{attribute 'GeneratedUsingTerminal: EK1122-0000-0018'}
{attribute addProperty BoxType "EK1122-0000-0018"}
{attribute addProperty Id "A_0060_AT2020_0250_0019_AT2020_0250A_0060_AT2020_0250_0019_AT2020_0250_29EE827680Beckhoff_AT2xxxsub_EK1100EK1100_1FC0878B2A_0001_AT2000_0233_0022AT2000_1809CD2F80A_0002_AT2000_0233_0023AT2000_1809CD2F80A_0003_AT2000_0233_0024AT2000_1809CD2F80A_0004_AT2000_0250_0016AT2000_2EA6C9BF84A_0005_AT2000_0250_0017AT2000_2EA6C9BF84A_0006_AT2000_0250_0018AT2000_2EA6C9BF84A_0007_AT2000_0250_0019AT2000_2EA6C9BF84A_0008_AT2000_0250_0020AT2000_2EA6C9BF84A_0009_AT2000_0250_0021AT2000_2EA6C9BF84A_0010_AT2000_0250_0022AT2000_2EA6C9BF84A_0011_AT2000_0250_0023AT2000_2EA6C9BF84A_0012_AT2001_0250_0016AT2001_2EA6C9BF84A_0013_AT2001_0250_0017AT2001_2EA6C9BF84A_0014_AT2001_0250_0018AT2001_2EA6C9BF84A_0015_AT2001_0250_0019AT2001_2EA6C9BF84A_0016_AT2001_0250_0020AT2001_2EA6C9BF84A_0017_AT2001_0250_0022AT2001_2EA6C9BF84A_0018_AT2001_0250_0023AT2001_2EA6C9BF84A_0019_AT2001_0250_0024AT2001_2EA6C9BF84A_0020_AT2002_0249_0021AT2002_2EA6C9BF84A_0021_AT2002_0249_0022AT2002_2EA6C9BF84A_0022_AT2002_0249_0023AT2002_2EA6C9BF84A_0023_AT2002_0250_0022AT2002_2EA6C9BF84A_0024_AT2002_0250_0023AT2002_2EA6C9BF84A_0025_AT2002_0250_0024AT2002_2EA6C9BF84A_0026_AT2020_0250_0018AT2020_2EA6C9BF84A_0027_AT2020_0250_0021AT2020_2EA6C9BF84A_0028_AT2021_0250_0018AT2021_2EA6C9BF84A_0029_AT2021_0250_0020AT2021_2EA6C9BF84A_0030_AT2025_0250_0018AT2025_2EA6C9BF84A_0031_AT2026_0250_0021AT2026_2EA6C9BF84A_0032_AT2026_0250_0023AT2026_2EA6C9BF84A_0033_AT2040_0250_0018AT2040_2EA6C9BF84A_0034_AT2040_0250_0019AT2040_2EA6C9BF84A_0035_AT2040_0250_0020AT2040_2EA6C9BF84A_0036_AT2040_0250_0021A_0036_AT2040_0250_0021_0B822AE480A_0037_AT2040_0250_0022A_0037_AT2040_0250_0022_033DCEC480A_0038_AT2040_0250_0023A_0038_AT2040_0250_0023_C339CA0C80A_0039_AT2040_0250_0024A_0039_AT2040_0250_0024_375958EA80A_0040_AT2041_0250_0018A_0040_AT2041_0250_0018_536500F280A_0041_AT2041_0250_0019A_0041_AT2041_0250_0019_F34F405680A_0042_AT2041_0250_0020A_0042_AT2041_0250_0020_5E65A51E80A_0043_AT2041_0250_0021A_0043_AT2041_0250_0021_AA0537F880A_0044_AT2041_0250_0022A_0044_AT2041_0250_0022_5A9A39BA80A_0045_AT2041_0250_0023A_0045_AT2041_0250_0023_51C662AC80A_0046_AT2042_0250_0024A_0046_AT2042_0250_0024_1B20CF3180A_0047_AT2050_0500_0016A_0047_AT2050_0500_0016_139F2B1180A_0048_AT2050_0500_0017A_0048_AT2050_0500_0017_3F977F4780A_0049_AT2050_0500_0018A_0049_AT2050_0500_0018_CBE655A880A_0050_AT2050_0500_0019A_0050_AT2050_0500_0019_15A3AE6F80A_0051_AT2050_0500_0020A_0051_AT2050_0500_0020_9B531B4E80A_0052_AT2050_0500_0021A_0052_AT2050_0500_0021_4516E08980A_0053_AT2050_0500_0022A_0053_AT2050_0500_0022_433BDDFE80A_0054_AT2050_0500_0023A_0054_AT2050_0500_0023_B2F2DF5580A_0055_AT2050_0500_0024A_0055_AT2050_0500_0024_8D42A08D80A_0056_AT2050_0501_0017A_0056_AT2050_0501_0017_A14AF4DB80A_0057_AT2050_0501_0020A_0057_AT2050_0501_0020_A9F510FB80A_0058_AT2050_0501_0021A_0058_AT2050_0501_0021_DD8E109080A_0061_AT2020_0250_0023_AT2020_0250A_0061_AT2020_0250_0023_AT2020_0250_2D9AB3DC80A_0062_AT2025_0250_0020_AT2025_0250A_0062_AT2025_0250_0020_AT2025_0250_8DB0F37880A_0063_AT2025_0250_0022_AT2025_0250A_0063_AT2025_0250_0022_AT2025_0250_E88F66A280A_0064_AT2025_0250_0023_AT2025_0250A_0064_AT2025_0250_0023_AT2025_0250_894F6FDC80A_0065_AT2026_0250_0019_AT2026_0250A_0065_AT2026_0250_0019_AT2026_0250_A5473B8A80A_0066_AT2026_0250_0020_AT2026_0250A_0066_AT2026_0250_0020_AT2026_0250_ADF8DFAA80A_0067_AT2026_0250_0022_AT2026_0250A_0067_AT2026_0250_0022_AT2026_0250_BF728FE680A_0068_AT2026_0250_0024_AT2026_0250A_0068_AT2026_0250_0024_AT2026_0250_71C0116580A_0069_AT2050_0501_0019_AT2050_0501A_0069_AT2050_0501_0019_AT2050_0501_10255FA680A_0070_AT2050_0501_0022_AT2050_0501A_0070_AT2050_0501_0022_AT2050_0501_E445CD4080A_0071_AT2050_0501_0023_AT2050_0501A_0071_AT2050_0501_0023_AT2050_0501_A5CC968480A_0072_AT2050_0501_0024_AT2050_0501A_0072_AT2050_0501_0024_AT2050_0501_05E6D62080"}
{attribute addProperty CRC "1138582487"}
{attribute addProperty Size "5810"}
TYPE Beckhoff_AT2xxxEK1122_43DD63D7 EXTENDS EK1122_1FC0878B :
STRUCT
	{attribute addProperty Name "A_0060_AT2020_0250_0019_AT2020_0250"}
	{attribute addProperty PreviousPort "Beckhoff AT2xxxEK1122 : D"}
	A_0060_AT2020_0250_0019_AT2020_0250 : A_0060_AT2020_0250_0019_AT2020_0250_29EE8276;
	{attribute addProperty Name "Beckhoff_AT2xxxsub_EK1100"}
	{attribute addProperty PreviousPort "A_0060(AT2020-0250-0019) (AT2020-0250) : C"}
	Beckhoff_AT2xxxsub_EK1100 : EK1100_1FC0878B;
	{attribute addProperty Name "A_0001_AT2000_0233_0022"}
	{attribute addProperty PreviousPort "Beckhoff AT2xxxsub EK1100 : C"}
	A_0001_AT2000_0233_0022 : AT2000_1809CD2F;
	{attribute addProperty Name "A_0002_AT2000_0233_0023"}
	{attribute addProperty PreviousPort "A_0001(AT2000-0233-0022) : C"}
	A_0002_AT2000_0233_0023 : AT2000_1809CD2F;
	{attribute addProperty Name "A_0003_AT2000_0233_0024"}
	{attribute addProperty PreviousPort "A_0002(AT2000-0233-0023) : C"}
	A_0003_AT2000_0233_0024 : AT2000_1809CD2F;
	{attribute addProperty Name "A_0004_AT2000_0250_0016"}
	{attribute addProperty PreviousPort "A_0003(AT2000-0233-0024) : C"}
	A_0004_AT2000_0250_0016 : AT2000_2EA6C9BF;
	{attribute addProperty Name "A_0005_AT2000_0250_0017"}
	{attribute addProperty PreviousPort "A_0004(AT2000-0250-0016) : C"}
	A_0005_AT2000_0250_0017 : AT2000_2EA6C9BF;
	{attribute addProperty Name "A_0006_AT2000_0250_0018"}
	{attribute addProperty PreviousPort "A_0005(AT2000-0250-0017) : C"}
	A_0006_AT2000_0250_0018 : AT2000_2EA6C9BF;
	{attribute addProperty Name "A_0007_AT2000_0250_0019"}
	{attribute addProperty PreviousPort "A_0006(AT2000-0250-0018) : C"}
	A_0007_AT2000_0250_0019 : AT2000_2EA6C9BF;
	{attribute addProperty Name "A_0008_AT2000_0250_0020"}
	{attribute addProperty PreviousPort "A_0007(AT2000-0250-0019) : C"}
	A_0008_AT2000_0250_0020 : AT2000_2EA6C9BF;
	{attribute addProperty Name "A_0009_AT2000_0250_0021"}
	{attribute addProperty PreviousPort "A_0008(AT2000-0250-0020) : C"}
	A_0009_AT2000_0250_0021 : AT2000_2EA6C9BF;
	{attribute addProperty Name "A_0010_AT2000_0250_0022"}
	{attribute addProperty PreviousPort "A_0009(AT2000-0250-0021) : C"}
	A_0010_AT2000_0250_0022 : AT2000_2EA6C9BF;
	{attribute addProperty Name "A_0011_AT2000_0250_0023"}
	{attribute addProperty PreviousPort "A_0010(AT2000-0250-0022) : C"}
	A_0011_AT2000_0250_0023 : AT2000_2EA6C9BF;
	{attribute addProperty Name "A_0012_AT2001_0250_0016"}
	{attribute addProperty PreviousPort "A_0011(AT2000-0250-0023) : C"}
	A_0012_AT2001_0250_0016 : AT2001_2EA6C9BF;
	{attribute addProperty Name "A_0013_AT2001_0250_0017"}
	{attribute addProperty PreviousPort "A_0012(AT2001-0250-0016) : C"}
	A_0013_AT2001_0250_0017 : AT2001_2EA6C9BF;
	{attribute addProperty Name "A_0014_AT2001_0250_0018"}
	{attribute addProperty PreviousPort "A_0013(AT2001-0250-0017) : C"}
	A_0014_AT2001_0250_0018 : AT2001_2EA6C9BF;
	{attribute addProperty Name "A_0015_AT2001_0250_0019"}
	{attribute addProperty PreviousPort "A_0014(AT2001-0250-0018) : C"}
	A_0015_AT2001_0250_0019 : AT2001_2EA6C9BF;
	{attribute addProperty Name "A_0016_AT2001_0250_0020"}
	{attribute addProperty PreviousPort "A_0015(AT2001-0250-0019) : C"}
	A_0016_AT2001_0250_0020 : AT2001_2EA6C9BF;
	{attribute addProperty Name "A_0017_AT2001_0250_0022"}
	{attribute addProperty PreviousPort "A_0016(AT2001-0250-0020) : C"}
	A_0017_AT2001_0250_0022 : AT2001_2EA6C9BF;
	{attribute addProperty Name "A_0018_AT2001_0250_0023"}
	{attribute addProperty PreviousPort "A_0017(AT2001-0250-0022) : C"}
	A_0018_AT2001_0250_0023 : AT2001_2EA6C9BF;
	{attribute addProperty Name "A_0019_AT2001_0250_0024"}
	{attribute addProperty PreviousPort "A_0018(AT2001-0250-0023) : C"}
	A_0019_AT2001_0250_0024 : AT2001_2EA6C9BF;
	{attribute addProperty Name "A_0020_AT2002_0249_0021"}
	{attribute addProperty PreviousPort "A_0019(AT2001-0250-0024) : C"}
	A_0020_AT2002_0249_0021 : AT2002_2EA6C9BF;
	{attribute addProperty Name "A_0021_AT2002_0249_0022"}
	{attribute addProperty PreviousPort "A_0020(AT2002-0249-0021) : C"}
	A_0021_AT2002_0249_0022 : AT2002_2EA6C9BF;
	{attribute addProperty Name "A_0022_AT2002_0249_0023"}
	{attribute addProperty PreviousPort "A_0021(AT2002-0249-0022) : C"}
	A_0022_AT2002_0249_0023 : AT2002_2EA6C9BF;
	{attribute addProperty Name "A_0023_AT2002_0250_0022"}
	{attribute addProperty PreviousPort "A_0022(AT2002-0249-0023) : C"}
	A_0023_AT2002_0250_0022 : AT2002_2EA6C9BF;
	{attribute addProperty Name "A_0024_AT2002_0250_0023"}
	{attribute addProperty PreviousPort "A_0023(AT2002-0250-0022) : C"}
	A_0024_AT2002_0250_0023 : AT2002_2EA6C9BF;
	{attribute addProperty Name "A_0025_AT2002_0250_0024"}
	{attribute addProperty PreviousPort "A_0024(AT2002-0250-0023) : C"}
	A_0025_AT2002_0250_0024 : AT2002_2EA6C9BF;
	{attribute addProperty Name "A_0026_AT2020_0250_0018"}
	{attribute addProperty PreviousPort "A_0025(AT2002-0250-0024) : C"}
	A_0026_AT2020_0250_0018 : AT2020_2EA6C9BF;
	{attribute addProperty Name "A_0027_AT2020_0250_0021"}
	{attribute addProperty PreviousPort "A_0026(AT2020-0250-0018) : C"}
	A_0027_AT2020_0250_0021 : AT2020_2EA6C9BF;
	{attribute addProperty Name "A_0028_AT2021_0250_0018"}
	{attribute addProperty PreviousPort "A_0027(AT2020-0250-0021) : C"}
	A_0028_AT2021_0250_0018 : AT2021_2EA6C9BF;
	{attribute addProperty Name "A_0029_AT2021_0250_0020"}
	{attribute addProperty PreviousPort "A_0028(AT2021-0250-0018) : C"}
	A_0029_AT2021_0250_0020 : AT2021_2EA6C9BF;
	{attribute addProperty Name "A_0030_AT2025_0250_0018"}
	{attribute addProperty PreviousPort "A_0029(AT2021-0250-0020) : C"}
	A_0030_AT2025_0250_0018 : AT2025_2EA6C9BF;
	{attribute addProperty Name "A_0031_AT2026_0250_0021"}
	{attribute addProperty PreviousPort "A_0030(AT2025-0250-0018) : C"}
	A_0031_AT2026_0250_0021 : AT2026_2EA6C9BF;
	{attribute addProperty Name "A_0032_AT2026_0250_0023"}
	{attribute addProperty PreviousPort "A_0031(AT2026-0250-0021) : C"}
	A_0032_AT2026_0250_0023 : AT2026_2EA6C9BF;
	{attribute addProperty Name "A_0033_AT2040_0250_0018"}
	{attribute addProperty PreviousPort "A_0032(AT2026-0250-0023) : C"}
	A_0033_AT2040_0250_0018 : AT2040_2EA6C9BF;
	{attribute addProperty Name "A_0034_AT2040_0250_0019"}
	{attribute addProperty PreviousPort "A_0033(AT2040-0250-0018) : C"}
	A_0034_AT2040_0250_0019 : AT2040_2EA6C9BF;
	{attribute addProperty Name "A_0035_AT2040_0250_0020"}
	{attribute addProperty PreviousPort "A_0034(AT2040-0250-0019) : C"}
	A_0035_AT2040_0250_0020 : AT2040_2EA6C9BF;
	{attribute addProperty Name "A_0036_AT2040_0250_0021"}
	{attribute addProperty PreviousPort "A_0035(AT2040-0250-0020) : C"}
	A_0036_AT2040_0250_0021 : A_0036_AT2040_0250_0021_0B822AE4;
	{attribute addProperty Name "A_0037_AT2040_0250_0022"}
	{attribute addProperty PreviousPort "A_0036(AT2040-0250-0021) : C"}
	A_0037_AT2040_0250_0022 : A_0037_AT2040_0250_0022_033DCEC4;
	{attribute addProperty Name "A_0038_AT2040_0250_0023"}
	{attribute addProperty PreviousPort "A_0037(AT2040-0250-0022) : C"}
	A_0038_AT2040_0250_0023 : A_0038_AT2040_0250_0023_C339CA0C;
	{attribute addProperty Name "A_0039_AT2040_0250_0024"}
	{attribute addProperty PreviousPort "A_0038(AT2040-0250-0023) : C"}
	A_0039_AT2040_0250_0024 : A_0039_AT2040_0250_0024_375958EA;
	{attribute addProperty Name "A_0040_AT2041_0250_0018"}
	{attribute addProperty PreviousPort "A_0039(AT2040-0250-0024) : C"}
	A_0040_AT2041_0250_0018 : A_0040_AT2041_0250_0018_536500F2;
	{attribute addProperty Name "A_0041_AT2041_0250_0019"}
	{attribute addProperty PreviousPort "A_0040(AT2041-0250-0018) : C"}
	A_0041_AT2041_0250_0019 : A_0041_AT2041_0250_0019_F34F4056;
	{attribute addProperty Name "A_0042_AT2041_0250_0020"}
	{attribute addProperty PreviousPort "A_0041(AT2041-0250-0019) : C"}
	A_0042_AT2041_0250_0020 : A_0042_AT2041_0250_0020_5E65A51E;
	{attribute addProperty Name "A_0043_AT2041_0250_0021"}
	{attribute addProperty PreviousPort "A_0042(AT2041-0250-0020) : C"}
	A_0043_AT2041_0250_0021 : A_0043_AT2041_0250_0021_AA0537F8;
	{attribute addProperty Name "A_0044_AT2041_0250_0022"}
	{attribute addProperty PreviousPort "A_0043(AT2041-0250-0021) : C"}
	A_0044_AT2041_0250_0022 : A_0044_AT2041_0250_0022_5A9A39BA;
	{attribute addProperty Name "A_0045_AT2041_0250_0023"}
	{attribute addProperty PreviousPort "A_0044(AT2041-0250-0022) : C"}
	A_0045_AT2041_0250_0023 : A_0045_AT2041_0250_0023_51C662AC;
	{attribute addProperty Name "A_0046_AT2042_0250_0024"}
	{attribute addProperty PreviousPort "A_0045(AT2041-0250-0023) : C"}
	A_0046_AT2042_0250_0024 : A_0046_AT2042_0250_0024_1B20CF31;
	{attribute addProperty Name "A_0047_AT2050_0500_0016"}
	{attribute addProperty PreviousPort "A_0046(AT2042-0250-0024) : C"}
	A_0047_AT2050_0500_0016 : A_0047_AT2050_0500_0016_139F2B11;
	{attribute addProperty Name "A_0048_AT2050_0500_0017"}
	{attribute addProperty PreviousPort "A_0047(AT2050-0500-0016) : C"}
	A_0048_AT2050_0500_0017 : A_0048_AT2050_0500_0017_3F977F47;
	{attribute addProperty Name "A_0049_AT2050_0500_0018"}
	{attribute addProperty PreviousPort "A_0048(AT2050-0500-0017) : C"}
	A_0049_AT2050_0500_0018 : A_0049_AT2050_0500_0018_CBE655A8;
	{attribute addProperty Name "A_0050_AT2050_0500_0019"}
	{attribute addProperty PreviousPort "A_0049(AT2050-0500-0018) : C"}
	A_0050_AT2050_0500_0019 : A_0050_AT2050_0500_0019_15A3AE6F;
	{attribute addProperty Name "A_0051_AT2050_0500_0020"}
	{attribute addProperty PreviousPort "A_0050(AT2050-0500-0019) : C"}
	A_0051_AT2050_0500_0020 : A_0051_AT2050_0500_0020_9B531B4E;
	{attribute addProperty Name "A_0052_AT2050_0500_0021"}
	{attribute addProperty PreviousPort "A_0051(AT2050-0500-0020) : C"}
	A_0052_AT2050_0500_0021 : A_0052_AT2050_0500_0021_4516E089;
	{attribute addProperty Name "A_0053_AT2050_0500_0022"}
	{attribute addProperty PreviousPort "A_0052(AT2050-0500-0021) : C"}
	A_0053_AT2050_0500_0022 : A_0053_AT2050_0500_0022_433BDDFE;
	{attribute addProperty Name "A_0054_AT2050_0500_0023"}
	{attribute addProperty PreviousPort "A_0053(AT2050-0500-0022) : C"}
	A_0054_AT2050_0500_0023 : A_0054_AT2050_0500_0023_B2F2DF55;
	{attribute addProperty Name "A_0055_AT2050_0500_0024"}
	{attribute addProperty PreviousPort "A_0054(AT2050-0500-0023) : C"}
	A_0055_AT2050_0500_0024 : A_0055_AT2050_0500_0024_8D42A08D;
	{attribute addProperty Name "A_0056_AT2050_0501_0017"}
	{attribute addProperty PreviousPort "A_0055(AT2050-0500-0024) : C"}
	A_0056_AT2050_0501_0017 : A_0056_AT2050_0501_0017_A14AF4DB;
	{attribute addProperty Name "A_0057_AT2050_0501_0020"}
	{attribute addProperty PreviousPort "A_0056(AT2050-0501-0017) : C"}
	A_0057_AT2050_0501_0020 : A_0057_AT2050_0501_0020_A9F510FB;
	{attribute addProperty Name "A_0058_AT2050_0501_0021"}
	{attribute addProperty PreviousPort "A_0057(AT2050-0501-0020) : C"}
	A_0058_AT2050_0501_0021 : A_0058_AT2050_0501_0021_DD8E1090;
	{attribute addProperty Name "A_0061_AT2020_0250_0023_AT2020_0250"}
	{attribute addProperty PreviousPort "Beckhoff AT2xxxEK1122 : B"}
	A_0061_AT2020_0250_0023_AT2020_0250 : A_0061_AT2020_0250_0023_AT2020_0250_2D9AB3DC;
	{attribute addProperty Name "A_0062_AT2025_0250_0020_AT2025_0250"}
	{attribute addProperty PreviousPort "A_0061(AT2020-0250-0023) (AT2020-0250) : C"}
	A_0062_AT2025_0250_0020_AT2025_0250 : A_0062_AT2025_0250_0020_AT2025_0250_8DB0F378;
	{attribute addProperty Name "A_0063_AT2025_0250_0022_AT2025_0250"}
	{attribute addProperty PreviousPort "A_0062(AT2025-0250-0020) (AT2025-0250) : C"}
	A_0063_AT2025_0250_0022_AT2025_0250 : A_0063_AT2025_0250_0022_AT2025_0250_E88F66A2;
	{attribute addProperty Name "A_0064_AT2025_0250_0023_AT2025_0250"}
	{attribute addProperty PreviousPort "A_0063(AT2025-0250-0022) (AT2025-0250) : C"}
	A_0064_AT2025_0250_0023_AT2025_0250 : A_0064_AT2025_0250_0023_AT2025_0250_894F6FDC;
	{attribute addProperty Name "A_0065_AT2026_0250_0019_AT2026_0250"}
	{attribute addProperty PreviousPort "A_0064(AT2025-0250-0023) (AT2025-0250) : C"}
	A_0065_AT2026_0250_0019_AT2026_0250 : A_0065_AT2026_0250_0019_AT2026_0250_A5473B8A;
	{attribute addProperty Name "A_0066_AT2026_0250_0020_AT2026_0250"}
	{attribute addProperty PreviousPort "A_0065(AT2026-0250-0019) (AT2026-0250) : C"}
	A_0066_AT2026_0250_0020_AT2026_0250 : A_0066_AT2026_0250_0020_AT2026_0250_ADF8DFAA;
	{attribute addProperty Name "A_0067_AT2026_0250_0022_AT2026_0250"}
	{attribute addProperty PreviousPort "A_0066(AT2026-0250-0020) (AT2026-0250) : C"}
	A_0067_AT2026_0250_0022_AT2026_0250 : A_0067_AT2026_0250_0022_AT2026_0250_BF728FE6;
	{attribute addProperty Name "A_0068_AT2026_0250_0024_AT2026_0250"}
	{attribute addProperty PreviousPort "A_0067(AT2026-0250-0022) (AT2026-0250) : C"}
	A_0068_AT2026_0250_0024_AT2026_0250 : A_0068_AT2026_0250_0024_AT2026_0250_71C01165;
	{attribute addProperty Name "A_0069_AT2050_0501_0019_AT2050_0501"}
	{attribute addProperty PreviousPort "A_0068(AT2026-0250-0024) (AT2026-0250) : C"}
	A_0069_AT2050_0501_0019_AT2050_0501 : A_0069_AT2050_0501_0019_AT2050_0501_10255FA6;
	{attribute addProperty Name "A_0070_AT2050_0501_0022_AT2050_0501"}
	{attribute addProperty PreviousPort "A_0069(AT2050-0501-0019) (AT2050-0501) : C"}
	A_0070_AT2050_0501_0022_AT2050_0501 : A_0070_AT2050_0501_0022_AT2050_0501_E445CD40;
	{attribute addProperty Name "A_0071_AT2050_0501_0023_AT2050_0501"}
	{attribute addProperty PreviousPort "A_0070(AT2050-0501-0022) (AT2050-0501) : C"}
	A_0071_AT2050_0501_0023_AT2050_0501 : A_0071_AT2050_0501_0023_AT2050_0501_A5CC9684;
	{attribute addProperty Name "A_0072_AT2050_0501_0024_AT2050_0501"}
	{attribute addProperty PreviousPort "A_0071(AT2050-0501-0023) (AT2050-0501) : C"}
	A_0072_AT2050_0501_0024_AT2050_0501 : A_0072_AT2050_0501_0024_AT2050_0501_05E6D620;
END_STRUCT
END_TYPE

(* stored: Version 1.2.0.0, ProductVersion 3.1.4024.9
   DUT Beckhoff_AT2xxxEK1122_43DD63D7: Id {6315a657-731a-4e66-818f-41e1f78a2ec3} *)
